(* IEC 61131-3 sources: AxisLib/src/Ar/MotionControl/AxisBasic, 6 files *)

(* ---- AxisBasic.typ ---- *)
(*
* File: AxisBasic.typ
* Copyright (c) 2023 Loupe
* https://loupe.team
*
* This file is part of AxisBasic, licensed under the MIT License.
*)

TYPE
	Configuration_typ : 	STRUCT
		Axis : ARRAY[0..MAI_MOTOR]OF AxisConfiguration_typ;
	END_STRUCT;
	AxisConfiguration_typ : 	STRUCT
		Active : BOOL;
		Power : BOOL;
	END_STRUCT;
	axisHmi_typ : 	STRUCT
		axis : ARRAY[0..MAI_MOTOR]OF axisHmiStatus_typ;
	END_STRUCT;
	axisHmiStatus_typ : 	STRUCT
		powered : BOOL;
		referenced : BOOL;
		active : BOOL;
	END_STRUCT;
END_TYPE

(* ---- AxisBasicCyclic.st ---- *)
(*
* File: AxisBasicCyclic.st
* Copyright (c) 2023 Loupe
* https://loupe.team
*
* This file is part of AxisBasic, licensed under the MIT License.
*)

PROGRAM _CYCLIC

	// Call PiperModuleInterface to interface with the rest of the machine
	PiperModuleInterface;

	// Call AxisBasicFn_Cyclic to control the axis
	FOR i:=0 TO MAI_MOTOR BY 1 DO

		IF Configuration.Axis[i].Active THEN

			IF homeAll THEN
				gMotorBasic[i].IN.CMD.Reference :=1;
			END_IF

			AxisBasicFn_Cyclic(gMotorBasic[i]);
			// Reset edge-sensitive gAxis commands set by HMI
			gMotorBasic[i].IN.CMD.MoveAbsolute := FALSE;
			gMotorBasic[i].IN.CMD.MoveAdditive := FALSE;
			gMotorBasic[i].IN.CMD.Halt := FALSE;
			gMotorBasic[i].IN.CMD.Stop := FALSE;
			gMotorBasic[i].IN.CMD.ClearReference := FALSE;
			gMotorBasic[i].IN.CMD.Reference := FALSE;
			// Error collection
			axisErrorCollector[i]();

			axisHmi.axis[i].active:=	gMotorBasic[i].OUT.Active;
			axisHmi.axis[i].powered:=	gMotorBasic[i].OUT.DriveStatus.ControllerStatus;
			axisHmi.axis[i].referenced:=gMotorBasic[i].OUT.Referenced;

		END_IF

	END_FOR

	homeAll:=0;

	//Homing check
	homeCheck(CLK := (gMachine.OUT.State = MACH_ST_RESETTING));
	IF homeCheck.Q THEN
		FOR i:=0 TO MAI_MOTOR BY 1 DO
			IF Configuration.Axis[i].Power AND NOT gMotorBasic[i].OUT.Referenced THEN
				errcolAddError(ADR(axisErrorCollector[i].ErrorSourceName),ADR('Axis not referenced'),0,0,gErrorCollector);
			END_IF

		END_FOR
	END_IF

END_PROGRAM

(* ---- AxisBasicInit.st ---- *)
(*
* File: AxisBasicInit.st
* Copyright (c) 2023 Loupe
* https://loupe.team
*
* This file is part of AxisBasic, licensed under the MIT License.
*)

PROGRAM _INIT

	// emptyPar is used to check for empty axis parameter structures
	brsmemset(ADR(emptyPar), 0, SIZEOF(emptyPar));

	// Initialize axes
	FOR i:=0 TO MAI_MOTOR BY 1 DO

		gMotorBasic[i].pAxisObject := ADR(gMotorNcm[i]);
		gMotorBasic[i].ErrorTextModuleName := 'acp10etxen';
		gMotorBasic[i].pEndlessPosition := ADR(gEndlessPosition[i]);

		// CFG
		gMotorBasic[i].IN.CFG.HomingMode:=		mcHOME_DEFAULT;

		gMotorBasic[i].IN.CFG.StopDeceleration:=	100000;

		// Only initialize parameters if they are empty
		IF( brsmemcmp(ADR(gMotorBasic[i].IN.PAR), ADR(emptyPar), SIZEOF(gMotorBasic[i].IN.PAR)) = 0 )THEN

			// Default parameters
			gMotorBasic[i].IN.PAR.Position:=			0;
			gMotorBasic[i].IN.PAR.Distance:=			0;
			gMotorBasic[i].IN.PAR.Direction:=			mcPOSITIVE_DIR;
			gMotorBasic[i].IN.PAR.Velocity:=			9000;
			gMotorBasic[i].IN.PAR.Acceleration:=		90000;
			gMotorBasic[i].IN.PAR.Deceleration:=		90000;

			gMotorBasic[i].IN.PAR.JogVelocity:=		2000;
			gMotorBasic[i].IN.PAR.JogAcceleration:=	20000;
			gMotorBasic[i].IN.PAR.JogDeceleration:=	20000;

		END_IF

		// Error collector
		axisErrorCollector[i].Axis := ADR(gMotorNcm[i]);
		axisErrorCollector[i].ErrorSourceName := 'Motor ';
		appendArrayIndex(i,ADR(axisErrorCollector[i].ErrorSourceName));
		axisErrorCollector[i].DataObjectName := 'acp10etxen';
		axisErrorCollector[i].pErrorCollector := ADR(gErrorCollector);
		axisErrorCollector[i].Enable := TRUE;

		// Expand Limit
		axisExpandLimit[i].Axis := ADR(gMotorNcm[i]);

	END_FOR

END_PROGRAM

(* ---- PiperModuleInterface.st ---- *)
(*
* File: PiperModuleInterface.st
* Copyright (c) 2023 Loupe
* https://loupe.team
*
* This file is part of AxisBasic, licensed under the MIT License.
*)

ACTION PiperModuleInterface:

	// Give this module a name so it is easier to debug
	ModuleInterface.ModuleName := 'Servo Manager';

	// Add a module to the Piper
	Module.ModuleInterface := ADR(ModuleInterface);
	Module.Piper := ADR(gMachine);
	Module();

	// Handle any machine states that this module needs to respond to
	CASE ModuleInterface.PiperState OF

		MACH_ST_BOOTING: // Wait for axes to come on line (NetworkInit) and restore position
			groupStatus := 1;
			ModuleInterface.ModuleStatus := 'Waiting on axis:';

			FOR i:=0 TO MAI_MOTOR BY 1 DO
				IF Configuration.Axis[i].Active THEN

					// Stay here if NOT(NetworkInit)
					IF NOT gMotorBasic[i].OUT.DriveStatus.NetworkInit THEN
						groupStatus := 0;
						ModuleInterface.ModuleStatus := CONCAT(ModuleInterface.ModuleStatus, CONCAT('Net-', CONCAT( CONCAT(tempStr, ':'), CONCAT(gMotorBasic[i].IN.CFG.Name, ' '))));
					END_IF

					IF NOT gMotorBasic[i].OUT.DataValid AND gSimulation THEN
						gMotorBasic[i].IN.CFG.HomingMode := mcHOME_DIRECT;
						gMotorBasic[i].IN.CMD.Reference := 1;

					END_IF;

					// Leave if currently OK and
					// no endless position is configured, data is invalid, OR homing is done
					groupStatus := groupStatus AND (	(gMotorBasic[i].pEndlessPosition = 0)
												OR	(gMotorBasic[i].OUT.DataValid = FALSE)
												OR	(gMotorBasic[i].OUT.DriveStatus.HomingOk) );

				END_IF
			END_FOR

			IF groupStatus THEN
				ModuleInterface.ModuleResponse:=	ModuleInterface.PiperState;
			END_IF

		//MACH_ST_STOPPED

		MACH_ST_RESETTING: // Power axes. Restore Position if appropriate

			CASE ModuleInterface.PiperSubState OF

				SUB_STATE_INIT:
					ModuleInterface.ModuleSubStateRequest:=	SUB_STATE_SERVO_POWER;

				SUB_STATE_SERVO_POWER:
					groupStatus := 1;
					ModuleInterface.ModuleStatus := 'Waiting on axis:';

					FOR i:=0 TO MAI_MOTOR BY 1 DO
						IF Configuration.Axis[i].Power THEN

							gMotorBasic[i].IN.CMD.Power := 1;

							IF NOT gMotorBasic[i].OUT.DriveStatus.ControllerStatus THEN
								groupStatus := 0;
								ModuleInterface.ModuleStatus := CONCAT(ModuleInterface.ModuleStatus, CONCAT(gMotorBasic[i].IN.CFG.Name, ' '));
							END_IF

						END_IF
					END_FOR

					IF groupStatus THEN

						ModuleInterface.ModuleResponse := ModuleInterface.PiperState;

					END_IF

			END_CASE

			//MACH_ST_IDLE:
			//MACH_ST_STARTING:
			//MACH_ST_EXECUTE:
			//MACH_ST_COMPLETING:
			//MACH_ST_COMPLETE:
			//MACH_ST_HOLDING:
			//MACH_ST_HELD:
			//MACH_ST_UNHOLDING:
			//MACH_ST_SUSPENDING:
			//MACH_ST_SUSPENDED:
			//MACH_ST_UNSUSPENDING:

		MACH_ST_ABORTING,
		MACH_ST_STOPPING: // Stop the axes if they are moving and power down

			CASE ModuleInterface.PiperSubState OF

				SUB_STATE_INIT:
					ModuleInterface.ModuleSubStateRequest:=	SUB_STATE_SERVO_STOP;

				SUB_STATE_SERVO_STOP:
					groupStatus := 1;
					ModuleInterface.ModuleStatus := 'Waiting on axis:';

					FOR i:=0 TO MAI_MOTOR BY 1 DO
						IF Configuration.Axis[i].Active THEN

							// Reset all move commands
							gMotorBasic[i].IN.CMD.Reference := 0;
							gMotorBasic[i].IN.CMD.MoveAbsolute := 0;
							gMotorBasic[i].IN.CMD.MoveAdditive := 0;
							gMotorBasic[i].IN.CMD.MoveVelocity := 0;
							gMotorBasic[i].IN.CMD.JogForward := 0;
							gMotorBasic[i].IN.CMD.JogReverse := 0;
							gMotorBasic[i].IN.CMD.MoveCyclicPosition := 0;
							gMotorBasic[i].IN.CMD.Halt := 0;

							// If you are moving, then stop
							gMotorBasic[i].IN.CMD.Stop := gMotorBasic[i].OUT.PLCOpenState.ContinuousMotion
							OR gMotorBasic[i].OUT.PLCOpenState.DiscreteMotion
							OR gMotorBasic[i].OUT.PLCOpenState.Homing
							OR gMotorBasic[i].OUT.PLCOpenState.SynchronizedMotion;

							IF gMotorBasic[i].IN.CMD.Stop OR gMotorBasic[i].OUT.PLCOpenState.Stopping THEN
								groupStatus := 0;
								ModuleInterface.ModuleStatus := CONCAT(ModuleInterface.ModuleStatus, CONCAT(gMotorBasic[i].IN.CFG.Name, ' '));
							END_IF

						END_IF
					END_FOR

					IF groupStatus THEN
						//If a drive is powered off (i.e. because of an error), we power everything off.
						powerOffRequired := FALSE;
						FOR i:= 0 TO MAI_MOTOR BY 1 DO
							IF ((Configuration.Axis[i].Active) AND (Configuration.Axis[i].Power) AND (NOT gMotorBasic[i].OUT.DriveStatus.ControllerStatus)) THEN
								powerOffRequired := TRUE;
							END_IF
						END_FOR
						//If we are in aborting we should also power off
						IF (ModuleInterface.PiperState = MACH_ST_ABORTING) OR (powerOffRequired) THEN
							ModuleInterface.ModuleSubStateRequest:=	SUB_STATE_SERVO_POWER_OFF;
						//If we are stopping we are done. Keep things powered
						ELSE
							ModuleInterface.ModuleResponse:=	ModuleInterface.PiperState;
						END_IF
					END_IF

				SUB_STATE_SERVO_POWER_OFF:
					groupStatus := 1;
					ModuleInterface.ModuleStatus := 'Waiting on axis:';

					FOR i:=0 TO MAI_MOTOR BY 1 DO
						IF Configuration.Axis[i].Power THEN

							gMotorBasic[i].IN.CMD.Power := 0;

							IF NOT(gMotorBasic[i].OUT.PLCOpenState.Disabled) THEN
								groupStatus := 0;
								ModuleInterface.ModuleStatus := CONCAT(ModuleInterface.ModuleStatus, CONCAT(gMotorBasic[i].IN.CFG.Name, ' '));
							END_IF

						END_IF
					END_FOR

					IF groupStatus THEN
						ModuleInterface.ModuleResponse:=	ModuleInterface.PiperState;
					END_IF

			END_CASE

		//MACH_ST_ABORTED,

		MACH_ST_CLEARING: // Check for axis ready to get out of clearing state
			groupStatus := 1;
			ModuleInterface.ModuleStatus := 'Waiting on axis:';

			FOR i:=0 TO MAI_MOTOR BY 1 DO
				IF Configuration.Axis[i].Active THEN

					IF (axisErrorCollector[i].Error
						OR NOT(gMotorBasic[i].OUT.DriveStatus.NetworkInit)
						OR NOT(gMotorBasic[i].OUT.DriveStatus.ControllerReady)
						) THEN
						groupStatus := 0;
						ModuleInterface.ModuleStatus := CONCAT(ModuleInterface.ModuleStatus, CONCAT(gMotorBasic[i].IN.CFG.Name, ' '));
					END_IF

					IF (axisErrorCollector[i].AxisError) THEN
						groupStatus := 0;
						ModuleInterface.ModuleStatus := CONCAT(ModuleInterface.ModuleStatus, CONCAT(gMotorBasic[i].IN.CFG.Name, ' '));
					END_IF

				END_IF
			END_FOR

			IF groupStatus THEN
				ModuleInterface.ModuleResponse := ModuleInterface.PiperState;
			END_IF

		MACH_ST_STOPPED:
			FOR i:=0 TO MAI_MOTOR BY 1 DO
				IF gMotorBasic[i].IN.CMD.Power AND NOT gMotorBasic[i].OUT.DriveStatus.ControllerStatus THEN
					gMachine.IN.CMD.Abort := TRUE;
				END_IF
			END_FOR
			ModuleInterface.ModuleResponse := ModuleInterface.PiperState;
			ModuleInterface.ModuleStatus := '';

		MACH_ST_ABORTED:

			ModuleInterface.ModuleResponse := ModuleInterface.PiperState;
			ModuleInterface.ModuleStatus := '';

			FOR i:=0 TO MAI_MOTOR BY 1 DO
				gMotorBasic[i].IN.CMD.Power := 0;
			END_FOR

		ELSE
			ModuleInterface.ModuleResponse := ModuleInterface.PiperState;
			ModuleInterface.ModuleStatus := '';

	END_CASE

	// Check for axis errors
	FOR i:=0 TO MAI_MOTOR BY 1 DO
		IF Configuration.Axis[i].Active THEN

			IF axisErrorCollector[i].AxisError AND gMotorBasic[i].OUT.DriveStatus.ControllerStatus THEN
				axisErrorCollector[i].Reset := TRUE;
				gMachine.IN.CMD.Stop := TRUE;
			ELSIF axisErrorCollector[i].AxisError AND NOT gMotorBasic[i].OUT.DriveStatus.ControllerStatus THEN
				axisErrorCollector[i].Reset := TRUE;
				gMachine.IN.CMD.Abort := TRUE;
			END_IF

		END_IF
	END_FOR

END_ACTION

(* ---- PiperModuleTemplate.var ---- *)
(*
* File: PiperModuleInterface.var
* Copyright (c) 2023 Loupe
* https://loupe.team
*
* This file is part of AxisBasic, licensed under the MIT License.
*)
VAR
	ModuleInterface : Module_Interface_typ;
	Module : Piper_Module_Fub;
END_VAR

(* ---- AxisBasic.var ---- *)
(*
* File: AxisBasic.var
* Copyright (c) 2023 Loupe
* https://loupe.team
*
* This file is part of AxisBasic, licensed under the MIT License.
*)
VAR
	axisHmi : axisHmi_typ := (0);
	axisErrorCollector : ARRAY[0..MAI_MOTOR] OF AxisAddErrorsToCollector;
	i : UDINT;
	emptyPar : AxisBasic_IN_PAR_typ;
	groupStatus : BOOL := FALSE; (*used to tell if the status of the group is all done*)
	powerOffRequired : BOOL;
	messageAdded : BOOL;
	noPistonHome : BOOL;
	Configuration : Configuration_typ;
	tempStr : STRING[512];
	axisExpandLimit : ARRAY[0..MAI_MOTOR] OF AxisExpandLimit;
END_VAR
